// TIA Portal V20 export
DATA_BLOCK "DB_PowerOn"   // DB462
// stored: AutoNumber false, InstanceOfName FB_PowerOn, InstanceOfType FB
"FB_PowerOn"
   // VAR
   //    sMachinePower : Bool;
   //    sMachineReadySoft : Bool;
   //    sOkForPowerON : Bool;
   //    sTimeMachineReadyDelay { S7_SetPoint := 'True'} : TON_TIME;
   //    sDelayPowerOFF { S7_SetPoint := 'True'} : TON_TIME;
   //    sDelayPowerON_1 { S7_SetPoint := 'True'} : TON_TIME;
   //    sDelayPowerON_2 { S7_SetPoint := 'True'} : TON_TIME;
   //    sX_AxisBrakeRelease { S7_SetPoint := 'True'} : Bool;
   //    sY_AxisBrakeRelease : Bool;
   //    sB_AxisBrakeRelease : Bool;
   // END_VAR
BEGIN
END_DATA_BLOCK
